# EPICS StreamDevice protocol: ESP8266/proto/lox02s.proto
OutTerminator = LF;

getOxygen{
        out "getOxygen";
        in "%f";
}
